// TIA Portal V19 export
DATA_BLOCK "WARNINGS"   // DB15
{ S7_Optimized_Access := 'FALSE' }
   VAR
      AIN { S7_SetPoint := 'True'} : Array[0.."MAX_AIN"] of "UDT_AINWARNS";   // AIN = 2 alarms/instance, 200 x 2 = 400 alarms, offset = 8000
      DIFF { S7_SetPoint := 'True'} : Array[0.."MAX_DIFF"] of "UDT_AINWARNS";   // DIFF = 2 alarms/instance, 200 x 2 = 400 alarms, offset = 8400
      Plant { S7_SetPoint := 'True'} : Array[0.."MAX_PLANT"] of "UDT_DINFAULTS";   // Plant = 1 alarm/instance, 24 x 8 (each type contains 8 instances) = 192 alarms, offset = 8800
   END_VAR
BEGIN
END_DATA_BLOCK
